Staubli VAL3: DebV2.pjx

--- DebV2.pjx ---
Parameters version=s7.4 stackSize=5000 millimeterUnit=true
Program file=Programmetest.pgx
Program file=start.pgx
Program file=stop.pgx
Data file=DebV2.dtx

--- DebV2.dtx ---
mdesc mNomSpeed
jointRx jJointRx[2]
  [1] = {j1=180}
dio SortiePower = {link=POWERLINK-1\%Q1}
dio EntreePower = {link=POWERLINK-1\%I0}
tool tTool = {z=50, fatherId=flange[0], ioLink=valve1}

--- start.pgx ---
program start()
begin
  call Programmetest()
end

--- Programmetest.pgx ---
program Programmetest()
begin
  wait(EntreePower==true)
  movej(jJointRx[0],tTool,mNomSpeed)
  movej(jJointRx[1],tTool,mNomSpeed)
  waitEndMove()
end
